FUNCTION F_Concat7 : T_MaxString
VAR_INPUT
	sOne : STRING;
	sTwo : STRING;
	sThree : STRING;
	sFour : STRING;
	sFive : STRING;
	sSix : STRING;
	sSeven : STRING;
END_VAR

F_Concat7 := CONCAT(
					sOne,
					F_Concat6( sTwo, sThree, sFour, sFive, sSix, sSeven )
				);

END_FUNCTION

(* stored: Version 1.1.0.1, ProductVersion 3.1.4022.9
   POU F_Concat7: Id {f5a0ea8d-1cd6-4e43-8618-dc4780fcdd37}, SpecialFunc None *)
